FUNCTION_BLOCK HardwareContainer
VAR
	// hardware control POUs
	m_crane: Crane;
	m_indic: ActivityIndicator(i_signalProcVar := EProcessVariables.Test_CraneFree);
	
	// products
	{attribute 'OPC.UA.DA' := '1'}
	{attribute 'OPC.UA.DA.Access' := '1'}
	m_craneWP: xPPUProduct(EProcessVariables.Crane_ProductType, EProcessVariables.Crane_ProductStamped);
	
	// hardware observation (if not included in hardware control)
	m_observeCrane: ObserveCrane(ADR(m_crane), ADR(m_craneWP));
	
	// control primitives
	m_craneMoveToStack: Crane_MoveToStack(ADR(m_crane));
	m_craneMoveToStamp: Crane_MoveToStamp(ADR(m_crane));
	m_craneMoveToLSC: Crane_MoveToLSC(ADR(m_crane));
	m_cranePickUpWP: Crane_PickUpWP(ADR(m_crane));
	m_cranePutDownWP: Crane_PutDownWP(ADR(m_crane));
	
	m_delay: Delay;
	m_indicCP_Crane: IndicateActivity(i_id := EPrimitives.Gen_IndicateActive_Crane, i_ptrIndicator := ADR(m_indic));
	m_forceVal_Crane: ForceProcessVariable(i_id := EPrimitives.Gen_ForceVariable_Crane);
	
	// module sequences
END_VAR

METHOD FB_init : BOOL
VAR_INPUT
	bInitRetains : BOOL; // if TRUE, the retain variables are initialized (warm start / cold start)
	bInCopyCode : BOOL;  // if TRUE, the instance afterwards gets moved into the copy code (online change)

	i_ptrStateTracker: POINTER TO StateTracker;
	i_ptrProcessManager: POINTER TO ProcessManager;
	
	i_ptrErrorManager: POINTER TO ErrorManagerBase;
END_VAR
m_craneMoveToStack.ProvideServices(i_ptrProcessManager, i_ptrStateTracker);
m_craneMoveToStamp.ProvideServices(i_ptrProcessManager, i_ptrStateTracker);
m_craneMoveToLSC.ProvideServices(i_ptrProcessManager, i_ptrStateTracker);
m_cranePickUpWP.ProvideServices(i_ptrProcessManager, i_ptrStateTracker);
m_cranePutDownWP.ProvideServices(i_ptrProcessManager, i_ptrStateTracker);

m_delay.ProvideServices(i_ptrProcessManager, i_ptrStateTracker);
m_indicCP_Crane.ProvideServices(i_ptrProcessManager, i_ptrStateTracker);
m_forceVal_Crane.ProvideServices(i_ptrProcessManager, i_ptrStateTracker);

// provide Behaviors to the Process Manager
i_ptrProcessManager^.AddPrimitive(ADR(m_craneMoveToStack));
i_ptrProcessManager^.AddPrimitive(ADR(m_craneMoveToStamp));
i_ptrProcessManager^.AddPrimitive(ADR(m_craneMoveToLSC));
i_ptrProcessManager^.AddPrimitive(ADR(m_cranePickUpWP));
i_ptrProcessManager^.AddPrimitive(ADR(m_cranePutDownWP));

i_ptrProcessManager^.AddPrimitive(ADR(m_delay));
i_ptrProcessManager^.AddPrimitive(ADR(m_indicCP_Crane));
i_ptrProcessManager^.AddPrimitive(ADR(m_forceVal_Crane));

// provide observations to the Process Manager
i_ptrStateTracker^.AddObservation(ADR(m_observeCrane));
i_ptrStateTracker^.AddObservation(ADR(m_indic));

// provide workpieces to the Process Manager
i_ptrStateTracker^.RegisterLocalProduct(EProducts.crane_product, ADR(m_craneWP));
END_METHOD

END_FUNCTION_BLOCK

(* stored: Version 1.1.0.1
   POU HardwareContainer: Id {da1cd6c3-75a3-4573-bc73-51d08569938e}, SpecialFunc None
   Method FB_init: Id {881a13a6-430f-4401-99e3-0a4ba74cb410} *)
